INTERFACE I_XtsHardware

PROPERTY DetectedNumberOfTracks : UINT
GET
END_GET
END_PROPERTY

PROPERTY ExpectedNumberOfParts : int
GET
END_GET
SET
END_SET
END_PROPERTY

PROPERTY ExpectedNumberOfTracks : int
GET
END_GET
SET
END_SET
END_PROPERTY

METHOD getAllMoversValid : BOOL
VAR_INPUT
END_VAR
END_METHOD

METHOD GetConfigMoverNumber : UDINT
VAR_INPUT
END_VAR
END_METHOD

METHOD GetDetectionState : DetectionStateEnum
VAR_INPUT
END_VAR
END_METHOD

METHOD getNumberMoversDetected : UDINT
VAR_INPUT
END_VAR
END_METHOD

METHOD GetTrackByNumber : I_XtsTrack
VAR_INPUT
	TrackNumber : UINT;
END_VAR
END_METHOD

METHOD GetTrackByOTCID : I_XtsTrack
VAR_INPUT
	trackOTCID : OTCID;
END_VAR
END_METHOD

METHOD HasXPU : BOOL
VAR_INPUT
END_VAR
END_METHOD

METHOD Is24VdcOK : HRESULT
VAR_INPUT
END_VAR
END_METHOD

METHOD Is48VdcOK : HRESULT
VAR_INPUT
END_VAR
END_METHOD

METHOD isExpectedMoversFound : BOOL
VAR_INPUT
END_VAR
END_METHOD

METHOD IsInitialised : BOOL
VAR_INPUT
END_VAR
END_METHOD

METHOD IsInSim : BOOL
VAR_INPUT
END_VAR
END_METHOD

PROPERTY MyName : string
GET
END_GET
END_PROPERTY

PROPERTY MyXpu : I_TcIoXtsProcessingUnit
GET
END_GET
SET
END_SET
END_PROPERTY

PROPERTY MyXts : INT
GET
END_GET
SET
END_SET
END_PROPERTY

METHOD RemoveTrackFromDetection : HRESULT
VAR_INPUT
	TrackToRemove : UINT;
END_VAR
END_METHOD

METHOD ResetParts : BOOL
END_METHOD

METHOD SetMoverNumbers : HRESULT
VAR_INPUT
	NumberOfMovers : INT;
END_VAR
END_METHOD

METHOD SetTrackForDetection : HRESULT
VAR_INPUT
	TrackToDetect : UINT;
END_VAR
END_METHOD

METHOD TriggerMoverDetection : HRESULT
VAR_INPUT
END_VAR
END_METHOD

METHOD TriggerMoverID : HRESULT
VAR_INPUT
END_VAR
END_METHOD

METHOD TriggerRedetection : HRESULT
VAR_INPUT
END_VAR
END_METHOD

END_INTERFACE

(* stored: Version 1.1.0.1
   Itf I_XtsHardware: Id {9afac880-0754-4de0-b157-657ea2ab2f5c}
   Folder Commands: Id {27c9da71-387e-4094-ae9a-f077ff9b1b1e}
   Folder Settings: Id {e3948c37-e7d1-40e0-b3aa-465d52d19205}
   Folder Status: Id {f56f8332-a404-49a0-b1fa-c3796e00575d}
   Property DetectedNumberOfTracks: Id {1f7b777e-4e84-4e05-a960-b4258ee4a093}
   Get Get: Id {b975fd9f-07a4-422f-a5dd-e3785eb793b3}
   Property ExpectedNumberOfParts: Id {8baf703f-4030-43b9-bdf8-f6888d62a51a}
   Get Get: Id {0b7c22e3-40c5-447c-8669-8bda14b6c107}
   Set Set: Id {5fd5e677-eecf-47de-bd59-50e6a5a429b3}
   Property ExpectedNumberOfTracks: Id {060a46c5-290c-4bcd-90e6-de762c9e2c08}
   Get Get: Id {32b0bf5c-9771-495a-89d6-3032bdd0b8c3}
   Set Set: Id {9407f136-b996-42ff-9b05-517db21ec39e}
   Method getAllMoversValid: Id {3d107ad0-1a72-4602-abbb-1177fad35523}
   Method GetConfigMoverNumber: Id {840a6c17-fbef-4810-9acd-02a47aa8f2b0}
   Method GetDetectionState: Id {fa37bb06-5333-4945-837b-ed2607a0f10b}
   Method getNumberMoversDetected: Id {f24c38ad-dbfa-488d-af77-9f21cd2a2d34}
   Method GetTrackByNumber: Id {fdddf6a5-daa4-4b5f-bc28-556a31f03729}
   Method GetTrackByOTCID: Id {32320bf3-efb9-473d-bca7-a0ced8f8657b}
   Method HasXPU: Id {4bb0c294-1f51-4661-82c9-c8d7d52811fe}
   Method Is24VdcOK: Id {d84db133-10f1-4c84-aee2-357bd38938fd}
   Method Is48VdcOK: Id {df545d44-305d-4b7a-922f-4b561f83d56a}
   Method isExpectedMoversFound: Id {aa48d66d-e689-4a24-808d-2ead7682c5a9}
   Method IsInitialised: Id {eb3371dd-7907-4a18-ba2b-9ef954004075}
   Method IsInSim: Id {5eeeddd9-9ad7-4819-b9a4-994a910fffac}
   Property MyName: Id {b43d0e80-e621-46e0-af70-0a677800dc98}
   Get Get: Id {494ebcb6-a0a6-498f-a4fa-49193344e0b2}
   Property MyXpu: Id {e2e815a3-d77a-4532-829a-eddabfcaecf8}
   Get Get: Id {bcee566b-b874-4152-ba22-6584fd88703d}
   Set Set: Id {98412ca9-12f3-48a0-a17f-85457d787566}
   Property MyXts: Id {53462daf-bea5-4a22-960f-7d5bfcc2ce3c}
   Get Get: Id {0d7e989b-6c34-4c03-ad75-2a4dfad812ae}
   Set Set: Id {09a1cb2a-649a-43ca-b93f-1edc829a7cd1}
   Method RemoveTrackFromDetection: Id {6b996083-6718-40f8-8385-c5509d71f04d}
   Method ResetParts: Id {1ef4fc6a-84af-4fb3-a74e-14a888b66822}
   Method SetMoverNumbers: Id {7821c5af-a98b-4e00-bdec-978858c91986}
   Method SetTrackForDetection: Id {e5174e94-1d43-416d-9cf0-82b8810737fe}
   Method TriggerMoverDetection: Id {3ca79f9d-8f1a-40ef-9b71-3df667743234}
   Method TriggerMoverID: Id {94d400e7-7631-41b8-b1e4-2b7514685c32}
   Method TriggerRedetection: Id {02f3159c-a37c-4b20-ae4e-7c65bf1966cb} *)
